INTERFACE IPAScaleTotalizing EXTENDS IPAScaleGravimetric

END_INTERFACE

(* stored: Version 1.1.0.1, ProductVersion 3.1.4020.12
   Itf IPAScaleTotalizing: Id {b8486f86-e96e-4a2d-903e-ab4fcd030a22} *)
